// TIA Portal V20 export
TYPE "UDT_RecepcionDeDispositivo"
   STRUCT
      Auxiliar_01 : UInt;
      Auxiliar_02 : UInt;
      Auxiliar_03 : UInt;
      ORDE : UInt;
      Protocolo { S7_SetPoint := 'True'} : "UDT_ProtocoloRecDispositivo";
   END_STRUCT;
END_TYPE
